// TIA Portal V16 export
// export: Created 2021-11-12T13:33:05.5900478Z, ExportSetting WithDefaults, DisplayName Totally Integrated Automation Portal, DisplayVersion V16 Update 3, DisplayName TIA Portal Version Control Interface, DisplayVersion V16 Update 2, DisplayName TIA Portal Openness, DisplayVersion V16 Update 3, DisplayName SINAMICS Startdrive Advanced, DisplayVersion V16 Update 5, DisplayName SINAMICS Startdrive G130, G150, S120, S150, SINAMICS MV, S210, DisplayVersion V16 Update 5, DisplayName SINAMICS Startdrive G110M, G120, G120C, G120D, G120P, G115D, DisplayVersion V16 Update 5, DisplayName STEP 7 Professional, DisplayVersion V16 Update 3, DisplayName STEP 7 Safety, DisplayVersion V16, DisplayName WinCC UA Professional, DisplayVersion V16 Update 3
DATA_BLOCK "STATUS_460"   // DB78
{ S7_Optimized_Access := 'TRUE' }
VERSION : 0.1
// stored: AutoNumber true, DBAccessibleFromOPCUA true, IsOnlyStoredInLoadMemory false, IsRetainMemResEnabled false, IsWriteProtectedInAS false, MemoryReserve 100
   VAR
      xxxxx___BinarySensors___xxxxx : Byte;
      "GL01-BG01" : Bool;   // Snímání pohybu dílu na dopravníku ++460+GL01 (M1)
      "GL02-BG01" : Bool;   // Snímání pohybu dílu na dopravníku ++460+GL02 (M3)
      "GL03-BG01" : Bool;   // Snímání pohybu dílu na dopravníku ++460+GL03 (M7.2)
      "GL04-BG01" : Bool;   // Snímání pohybu dílu na dopravníku ++460+GL04 (M5)
      "UC21-FC01_14" : Bool;   // 400V Dopravník ++460 OK
      "UC21-FC02_14" : Bool;   // 400V Dopravník ++460 OK
      "UC21-FC03_14" : Bool;   // 400V Dopravník ++460 OK
      "UC21-FC04_14" : Bool;   // 400V Dopravník ++460 OK
      xxxxx___BinaryOthers___xxxxx : Byte;
      "UH31-SF07_14" : Bool;   // Conveyor GL01 Remote
      "UH11-SF01_14" : Bool;   // Conveyor Remote
      UH31_SF07_24 : Bool;   // Conveyor GL01 Automat
      "UH11-SF01_24" : Bool;   // Conveyor Automat
      "UH31-SF09_14" : Bool;   // Conveyor GL01 Start automat
      "UH11-SF03_14" : Bool;   // Conveyor Start automat
      "UH31-SF10_12" : Bool;   // Conveyor GL01 Stop
      "UH11-SF04_12" : Bool;   // Conveyor Stop
      "UH31-SF08_14" : Bool;   // Conveyor GL01 Manual Backward
      "UH31-SF08_24" : Bool;   // Conveyor GL01 Manual Forward
      "UH11-SF05_14" : Bool;   // Conveyor GL02 Manual Backward
      "UH11-SF05_24" : Bool;   // Conveyor GL02 Manual Forward
      "UH11-SF06_14" : Bool;   // Conveyor GL03 Manual Backward
      "UH11-SF06_24" : Bool;   // Conveyor GL03 Manual Forward
      "UH11-SF07_14" : Bool;   // Conveyor GL04 Manual Backward
      "UH11-SF07_24" : Bool;   // Conveyor GL04 Manual Forward
      "UH11-SF08_14" : Bool;   // Bedna Žádost o výměnu
      "UH11-SF09_14" : Bool;   // Bedna vyměněna
      "UH31-SF11_X2" : Bool;   // Dopravník GL01 - blokování pásu v kleci
      xxxxx___Drives___xxxxx : Byte;
      "GL01-MA01" : Struct   // Conveyour to blasting machine (M1) - motor / Dopravník ke tryskači (M1) - motor
         Main : "UDT_Status_main";
         Specific : "UDT_Drive1_Status_specific";
         Error : "UDT_Error01";
      END_STRUCT;
      "GL02-MA01" : Struct   // Conveyour to blasting machine (M3) - motor / Dopravník ke tryskači (M3) - motor
         Main : "UDT_Status_main";
         Specific : "UDT_Drive1_Status_specific";
         Error : "UDT_Error01";
      END_STRUCT;
      "GL03-MA01" : Struct   // Conveyour to blasting machine (M7.2) - motor / Dopravník ke tryskači (M7.2) - motor
         Main : "UDT_Status_main";
         Specific : "UDT_Drive1_Status_specific";
         Error : "UDT_Error01";
      END_STRUCT;
      "GL04-MA01" : Struct   // Conveyour to blasting machine (M5) - motor / Dopravník ke tryskači (M5) - motor
         Main : "UDT_Status_main";
         Specific : "UDT_Drive1_Status_specific";
         Error : "UDT_Error01";
      END_STRUCT;
      "UC21-TA01" : Struct   // Conveyour to blasting machine (M1) - G120 / Dopravník ke tryskači (M1) - měnič G120
         Main : "UDT_Status_main";
         Specific : "UDT_SINAMICS_G120_Status_specific";
         Error : "UDT_Error02";
      END_STRUCT;
      "UC21-TA02" : Struct   // Conveyour to blasting machine (M3) - G120 / Dopravník ke tryskači (M3) - měnič G120
         Main : "UDT_Status_main";
         Specific : "UDT_SINAMICS_G120_Status_specific";
         Error : "UDT_Error02";
      END_STRUCT;
      "UC21-TA03" : Struct   // Conveyour to blasting machine (M7.2) - G120 / Dopravník ke tryskači (M7.2) - měnič G120
         Main : "UDT_Status_main";
         Specific : "UDT_SINAMICS_G120_Status_specific";
         Error : "UDT_Error02";
      END_STRUCT;
      "UC21-TA04" : Struct   // Conveyour to blasting machine (M5) - G120 / Dopravník ke tryskači (M5) - měnič G120
         Main : "UDT_Status_main";
         Specific : "UDT_SINAMICS_G120_Status_specific";
         Error : "UDT_Error02";
      END_STRUCT;
      xxxxx___Others___xxxxx : Byte;
      CL01 : Struct   // Box - parts not blasted / Bedna na neotryskané kusy
         Main : "UDT_Status_main";
         Specific { S7_SetPoint := 'True'} : "UDT_PartCounter_Status";
         Error { S7_SetPoint := 'True'} : "UDT_Error01";
      END_STRUCT;
      xxxxx___Alarms___xxxxx : Byte;
      CL01_Warn : Struct   // CL01 - box full / CL01 - bedna plná.
         Main : "UDT_Status_main";
         Specific { S7_SetPoint := 'True'} : "UDT_DI_Mon_Status_specific";
         Error { S7_SetPoint := 'True'} : "UDT_Error01";
      END_STRUCT;
      CL01_Alarm : Struct   // CL01 - box full / CL01 - bedna plná.
         Main : "UDT_Status_main";
         Specific : "UDT_DI_Mon_Status_specific";
         Error : "UDT_Error01";
      END_STRUCT;
   END_VAR
BEGIN
END_DATA_BLOCK
